Fanuc KAREL source: kb00020.KL

PROGRAM KB00020
%STACKSIZE=65535
%PRIORITY=65535
%NOLOCKGROUP
VAR
P1 : INTEGER
RESULT : STRING[80]
BEGIN
P1=1
-- UNRESOLVED_PC line 8 opcodes [27 22 76 75] marker_code=12
END KB00020
